# B&R Automation Studio project dbserv_0640 (part 6)

```c
				/* =========================================================== */
				/* DFA-Zustand: Datenobjekt für Datenpunktdefinitionen löschen */
				/* =========================================================== */
				case cCD_PARSER_STATE_DEL_DO_POINT:
					iDatObjDelete.enable = TRUE;
					iDatObjDelete.ident = iDatObjInfo.ident;
					DatObjDelete(&iDatObjDelete);
					if (iDatObjDelete.status == 0) {
						ParserState = cCD_PARSER_STATE_CREATE_DO_POINT;
					}
					else if (iDatObjDelete.status != ERR_FUB_BUSY) {
						ParserState = cCD_PARSER_STATE_ERROR;
					}
					break;

				/* =========================================================== */
				/* DFA-Zustand: Datenobjekt für Datenpunktdefinitionen anlegen */
				/* =========================================================== */
				case cCD_PARSER_STATE_CREATE_DO_POINT:
					iDatObjCreate.enable = TRUE;
					iDatObjCreate.grp = 0;
					iDatObjCreate.pName = (unsigned long)"DpDesc";
					iDatObjCreate.len = countDefinedPoint * sizeof(POINT_DESC);
					iDatObjCreate.MemType = doUSRRAM;
					iDatObjCreate.Option = !doNO_CS;
					iDatObjCreate.pCpyData = (unsigned long)pPointDesc;
					DatObjCreate(&iDatObjCreate);
					if (iDatObjCreate.status == 0) {
						ParserState = cCD_PARSER_STATE_ALLOC_ACCESS_DATA;
					}
					else if (iDatObjCreate.status != ERR_FUB_BUSY) {
						ParserState = cCD_PARSER_STATE_ERROR;
					}
					break;

				/* ======================================= */
				/* DFA-Zustand: Zählen der DBS-Datenpunkte */
				/* ======================================= */
				case cCD_PARSER_STATE_ALLOC_ACCESS_DATA:

					/* --------------------------------------- */
					/* Speicher für Datentypzugriff allokieren */
					/* --------------------------------------- */
					memSize = 0;
					for (i=0; i<=maxDbsUnit; i++) {
						if (pAccessUnit[i].countType > 0) {
							memSize += pAccessUnit[i].countType;
						}
					}
					memSize *= sizeof(ACCESS_TYPE);
					StateTMP_alloc = TMP_alloc(memSize, (void*)&pAccessType);
					if (StateTMP_alloc == 0) {
						SmemSize += 0;
						StmpSize += memSize;
						memset(pAccessType, 0, memSize);

						/* ------------------------------------------ */
						/* Speicher für Anlagenzugriff initialisieren */
						/* ------------------------------------------ */
						pAccessTypeWork = pAccessType;
						for (i=0; i<=maxDbsUnit; i++) {
							if (pAccessUnit[i].countType > 0) {
								pAccessUnit[i].pAccessType = pAccessTypeWork;
								pAccessTypeWork += pAccessUnit[i].countType;
							}
						}

						/* ------------------------------------------- */
						/* Speicher für Datentypzugriff initialisieren */
						/* ------------------------------------------- */
						for (i=0; i<countDefinedPoint; i++) {
							DbsUnit = pPointDesc[i].dbsUnit;
							DbsType = pPointDesc[i].dbsType;
							DbsPoint = pPointDesc[i].dbsPoint;
							pAccessUnit[DbsUnit].pAccessType[DbsType].countPoint = (DbsPoint + 1 > pAccessUnit[DbsUnit].pAccessType[DbsType].countPoint) ? DbsPoint + 1 : pAccessUnit[DbsUnit].pAccessType[DbsType].countPoint;
							pTypeDesc[DbsType].countRelatedPoints++;
						}

						/* ----------------------------------------- */
						/* Speicher für Datenpunktzugriff allokieren */
						/* ----------------------------------------- */
						memSize = 0;
						for (i=0; i<=maxDbsUnit; i++) {
							if (pAccessUnit[i].pAccessType != NULL) {
								for (j=0; j<pAccessUnit[i].countType; j++) {
									memSize += pAccessUnit[i].pAccessType[j].countPoint;
								}
							}
						}
						memSize *= sizeof(ACCESS_POINT);
						StateTMP_alloc = TMP_alloc(memSize, (void*)&pAccessPoint);
						if (StateTMP_alloc == 0) {
							SmemSize += 0;
							StmpSize += memSize;
							memset(pAccessPoint, 0, memSize);

							/* ------------------------------------------- */
							/* Speicher für Datentypzugriff initialisieren */
							/* ------------------------------------------- */
							pAccessPointWork = pAccessPoint;
							for (i=0; i<=maxDbsUnit; i++) {
								for (j=0; j<pAccessUnit[i].countType; j++) {
									if (pAccessUnit[i].pAccessType[j].countPoint > 0) {
										pAccessUnit[i].pAccessType[j].pAccessPoint = pAccessPointWork;
										pAccessPointWork = pAccessPointWork + pAccessUnit[i].pAccessType[j].countPoint;
									}
								}
							}

							/* --------------------------------------------- */
							/* Speicher für Datenpunktzugriff initialisieren */
							/* --------------------------------------------- */
							pAccessDataWork = NULL;
							for (i=0; i<countDefinedPoint; i++) {
								DbsUnit = pPointDesc[i].dbsUnit;
								DbsType = pPointDesc[i].dbsType;
								DbsPoint = pPointDesc[i].dbsPoint;
								countItem = pTypeDesc[DbsType].countItem;
								countTimeItem = pTypeDesc[DbsType].countTimeItem;

								pAccessUnit[DbsUnit].pAccessType[DbsType].pAccessPoint[DbsPoint].pAccessData = pAccessDataWork;
								pAccessTypeWork = &pAccessUnit[DbsUnit].pAccessType[DbsType];
								len = 0;

								pAccessTypeWork->offExtern = len;
								pAccessTypeWork->lenExtern = pTypeDesc[DbsType].sizeType;
								len = pAccessTypeWork->lenExtern;
								if (len % 2 != 0) len++;

								pAccessTypeWork->offIntern = pAccessTypeWork->offExtern + len;
								pAccessTypeWork->lenIntern = pTypeDesc[DbsType].sizeIntType;
								len = pAccessTypeWork->lenIntern;
								if (len % 2 != 0) len++;

								pAccessTypeWork->offiExtern = pAccessTypeWork->offIntern + len;
								pAccessTypeWork->leniExtern = pTypeDesc[DbsType].sizeType;
								pAccessTypeWork->leniExternAlign = (pAccessTypeWork->leniExtern > 1 && pAccessTypeWork->leniExtern % 2 != 0) ? pAccessTypeWork->leniExtern + 1 : pAccessTypeWork->leniExtern;
								pAccessTypeWork->leniExternNext = pAccessTypeWork->leniExternAlign;
								len = countEventInstance * pAccessTypeWork->leniExternAlign;
								if (len % 2 != 0) len++;

								pAccessTypeWork->offValid = pAccessTypeWork->offiExtern + len;
								pAccessTypeWork->lenValid = sizeof(ACCESS_ITEM_VALID);
								pAccessTypeWork->lenValidAlign = (pAccessTypeWork->lenValid > 1 && pAccessTypeWork->lenValid % 2 != 0) ? pAccessTypeWork->lenValid + 1 : pAccessTypeWork->lenValid;
								len = countItem * pAccessTypeWork->lenValidAlign;
								if (len % 2 != 0) len++;

								pAccessTypeWork->offTime = pAccessTypeWork->offValid + len;
								pAccessTypeWork->lenTime = sizeof(RTCtime_typ);
								pAccessTypeWork->lenTimeAlign = (pAccessTypeWork->lenTime > 1 && pAccessTypeWork->lenTime % 2 != 0) ? pAccessTypeWork->lenTime + 1 : pAccessTypeWork->lenTime;
								len = countItem * pAccessTypeWork->lenTimeAlign;
								if (len % 2 != 0) len++;

								pAccessTypeWork->offiTime = pAccessTypeWork->offTime + len;
								pAccessTypeWork->leniTime = sizeof(RTCtime_typ);
								pAccessTypeWork->leniTimeAlign = (pAccessTypeWork->leniTime > 1 && pAccessTypeWork->leniTime % 2 != 0) ? pAccessTypeWork->leniTime + 1 : pAccessTypeWork->leniTime;
								pAccessTypeWork->leniTimeNext = countItem * pAccessTypeWork->leniTimeAlign;
								len = countEventInstance * pAccessTypeWork->leniTimeNext;
								if (len % 2 != 0) len++;

								pAccessTypeWork->offWritelink = pAccessTypeWork->offiTime + len;
								pAccessTypeWork->lenWritelink = sizeof(ACCESS_ITEM_WRITE_LINK);
								pAccessTypeWork->lenWritelinkAlign = (pAccessTypeWork->lenWritelink > 1 && pAccessTypeWork->lenWritelink % 2 != 0) ? pAccessTypeWork->lenWritelink + 1 : pAccessTypeWork->lenWritelink;
								len = countItem * pAccessTypeWork->lenWritelinkAlign;
								if (len % 2 != 0) len++;

								pAccessTypeWork->offWritehandle = pAccessTypeWork->offWritelink + len;
								pAccessTypeWork->lenWritehandle = sizeof(ACCESS_ITEM_WRITE_HANDLE);
								pAccessTypeWork->lenWritehandleAlign = (pAccessTypeWork->lenWritehandle > 1 && pAccessTypeWork->lenWritehandle % 2 != 0) ? pAccessTypeWork->lenWritehandle + 1 : pAccessTypeWork->lenWritehandle;
								len = countItem * pAccessTypeWork->lenWritehandleAlign;
								if (len % 2 != 0) len++;

								pAccessTypeWork->offiEventlink = pAccessTypeWork->offWritehandle + len;
								pAccessTypeWork->leniEventlink = sizeof(ACCESS_ITEM_EVENT_LINK);
								pAccessTypeWork->leniEventlinkAlign = (pAccessTypeWork->leniEventlink > 1 && pAccessTypeWork->leniEventlink % 2 != 0) ? pAccessTypeWork->leniEventlink + 1 : pAccessTypeWork->leniEventlink;
								pAccessTypeWork->leniEventlinkNext = countItem * pAccessTypeWork->leniEventlinkAlign;
								len = countEventInstance * pAccessTypeWork->leniEventlinkNext;
								if (len % 2 != 0) len++;

								pAccessTypeWork->offiReleasestream = pAccessTypeWork->offiEventlink + len;
								pAccessTypeWork->leniReleasestream = sizeof(ACCESS_ITEM_RELEASE);
								pAccessTypeWork->leniReleasestreamAlign = (pAccessTypeWork->leniReleasestream > 1 && pAccessTypeWork->leniReleasestream % 2 != 0) ? pAccessTypeWork->leniReleasestream + 1 : pAccessTypeWork->leniReleasestream;
								pAccessTypeWork->leniReleasestreamNext = countItem * pAccessTypeWork->leniReleasestreamAlign;
								len = countEventInstance * pAccessTypeWork->leniReleasestreamNext;
								if (len % 2 != 0) len++;

								pAccessTypeWork->offiHyst = pAccessTypeWork->offiReleasestream + len;
								pAccessTypeWork->leniHyst = pTypeDesc[DbsType].sizeType;
								pAccessTypeWork->leniHystAlign = (pAccessTypeWork->leniHyst > 1 && pAccessTypeWork->leniHyst % 2 != 0) ? pAccessTypeWork->leniHyst + 1 : pAccessTypeWork->leniHyst;
								pAccessTypeWork->leniHystNext = pAccessTypeWork->leniHystAlign;
								len = countEventInstance * pAccessTypeWork->leniHystNext;
								if (len % 2 != 0) len++;

								pAccessTypeWork->offiEvent = pAccessTypeWork->offiHyst + len;
								pAccessTypeWork->leniEvent = sizeof(ACCESS_ITEM_EVENT_STATE);
								pAccessTypeWork->leniEventAlign = (pAccessTypeWork->leniEvent > 1 && pAccessTypeWork->leniEvent % 2 != 0) ? pAccessTypeWork->leniEvent + 1 : pAccessTypeWork->leniEvent;
								pAccessTypeWork->leniEventNext = countItem * pAccessTypeWork->leniEventAlign;
								len = countEventInstance * pAccessTypeWork->leniEventNext;
								if (len % 2 != 0) len++;

								pAccessTypeWork->offFubInstance = pAccessTypeWork->offiEvent + len;
								pAccessTypeWork->lenFubInstance = sizeof(ACCESS_FUB_INSTANCE);
								pAccessTypeWork->lenFubInstanceAlign = (pAccessTypeWork->lenFubInstance > 1 && pAccessTypeWork->lenFubInstance % 2 != 0) ? pAccessTypeWork->lenFubInstance + 1 : pAccessTypeWork->lenFubInstance;
								len = countItem * pAccessTypeWork->lenFubInstanceAlign;
								if (len % 2 != 0) len++;

								pAccessDataWork = (ACCESS_DATA*)((unsigned char*)pAccessDataWork + pAccessTypeWork->offFubInstance + len);
							} /* (i=0; i<countDefinedPoint; i++) */

							/* ---------------- */
							/* nächster Zustand */
							/* ---------------- */
							ParserState = cCD_PARSER_STATE_COMPARE_DO_DATA;

						} /* (StateTMP_alloc == 0) */
						else {
							/* Fehler bei TMP_alloc */
							ParserState = cCD_PARSER_STATE_ERROR;
						}
					} /* (StateTMP_alloc == 0) */
					else {
						/* Fehler bei TMP_alloc */
						ParserState = cCD_PARSER_STATE_ERROR;
					}
					break;

				/* ==================================== */
				/* DFA-Zustand: Datenobjekt vorhanden ? */
				/* ==================================== */
				case cCD_PARSER_STATE_COMPARE_DO_DATA:
					memSize = (unsigned long)pAccessDataWork;
					if (DbsMemTypeData == 0) {
						StateTMP_alloc = TMP_alloc(memSize, (void*)&pAccessData);
						if (StateTMP_alloc == 0) {
							SmemSize += 0;
							StmpSize += memSize;
							memset(pAccessData, 0, memSize);
							ParserState = cCD_PARSER_STATE_WORK_DATA;
						}
						else {
							ParserState = cCD_PARSER_STATE_ERROR;
						}
					}
					else {
						iDatObjInfo.enable = TRUE;
						iDatObjInfo.pName = (unsigned long)"dbsData";
						DatObjInfo(&iDatObjInfo);
						if (iDatObjInfo.status == 0) {
							/* Datenmodul-Alignment beachten */
							if (iDatObjInfo.len >= memSize &&
								iDatObjInfo.len <  memSize + sizeof(unsigned long) &&
								DbsTypeChanged  == FALSE &&
								DbsPointChanged == FALSE)
							{
								pAccessData = (ACCESS_DATA*)iDatObjInfo.pDatObjMem;
								ParserState = cCD_PARSER_STATE_WORK_DATA;
							}
							else {
								ParserState = cCD_PARSER_STATE_DEL_DO_DATA;
							}
						}
						else if (iDatObjInfo.status == doERR_MODULNOTFOUND) {
							ParserState = cCD_PARSER_STATE_CREATE_DO_DATA;
						}
						else if (iDatObjInfo.status != ERR_FUB_BUSY) {
							ParserState = cCD_PARSER_STATE_ERROR;
						}
					}
					break;

				/* ================================ */
				/* DFA-Zustand: Datenobjekt löschen */
				/* ================================ */
				case cCD_PARSER_STATE_DEL_DO_DATA:
					iDatObjDelete.enable = TRUE;
					iDatObjDelete.ident = iDatObjInfo.ident;
					DatObjDelete(&iDatObjDelete);
					if (iDatObjDelete.status == 0) {
						ParserState = cCD_PARSER_STATE_CREATE_DO_DATA;
					}
					else if (iDatObjDelete.status != ERR_FUB_BUSY) {
						ParserState = cCD_PARSER_STATE_ERROR;
					}
					break;

				/* ==================================== */
				/* DFA-Zustand: Datenobjekt neu anlegen */
				/* ==================================== */
				case cCD_PARSER_STATE_CREATE_DO_DATA:
					iDatObjCreate.enable = TRUE;
					iDatObjCreate.grp = 0;
					iDatObjCreate.pName = (unsigned long)"dbsData";
					iDatObjCreate.len = memSize;
					iDatObjCreate.MemType = doUSRRAM;
					iDatObjCreate.Option = doNO_CS;
					iDatObjCreate.pCpyData = NULL;
					DatObjCreate(&iDatObjCreate);
					if (iDatObjCreate.status == 0) {
						pAccessData = (ACCESS_DATA*)iDatObjCreate.pDatObjMem;
						SmemSize += 0;
						StmpSize += memSize;
						memset(pAccessData, 0, memSize);
						ParserState = cCD_PARSER_STATE_WORK_DATA;
					}
					else if (iDatObjCreate.status != ERR_FUB_BUSY) {
						ParserState = cCD_PARSER_STATE_ERROR;
					}
					break;

				/* ======================================= */
				/* DFA-Zustand: Zählen der DBS-Datenpunkte */
				/* ======================================= */
				case cCD_PARSER_STATE_WORK_DATA:

					/* ------------------------------ */
					/* Pointer auf Datenpunkte setzen */
					/* ------------------------------ */
					for (i=0; i<countDefinedPoint; i++) {
						DbsUnit = pPointDesc[i].dbsUnit;
						DbsType = pPointDesc[i].dbsType;
						DbsPoint = pPointDesc[i].dbsPoint;
						pAccessUnit[DbsUnit].pAccessType[DbsType].pAccessPoint[DbsPoint].pAccessData += (unsigned long)pAccessData;
					}

					/* ---------------------- */
					/* Fubinstanzen eintragen */
					/* ---------------------- */
					for (i=0; i<countFubInstance; i++) {
						DbsUnit = pFubInstanceDesc[i].dbsUnit;
						DbsType = pFubInstanceDesc[i].dbsType;
						DbsPoint = pFubInstanceDesc[i].dbsPoint;
						DbsItem = pFubInstanceDesc[i].dbsItem;
						pAccessTypeWork  = &pAccessUnit[DbsUnit].pAccessType[DbsType];
						pAccessPointWork = &pAccessUnit[DbsUnit].pAccessType[DbsType].pAccessPoint[DbsPoint];
						pAccessFubInstance = (USINT**)(pAccessPointWork->pAccessData + pAccessTypeWork->offFubInstance + DbsItem * pAccessTypeWork->lenFubInstanceAlign);
						*pAccessFubInstance = pFubInstanceDesc[i].pFubInstance;
					}

					/* ---------------- */
					/* nächster Zustand */
					/* ---------------- */
					ParserState = cCD_PARSER_STATE_COMPARE_DO_EVENT;
					break;

				/* ==================================== */
				/* DFA-Zustand: Datenobjekt vorhanden ? */
				/* ==================================== */
				case cCD_PARSER_STATE_COMPARE_DO_EVENT:
					memSize = (maxDbsType + 1) * sizeof(ACCESS_EVENT_PIPE);
					for (i=0; i<=maxDbsType; i++) {
						if (pTypeDesc[i].pItemDesc != NULL && pTypeDesc[i].countRelatedPoints > 0) {
							memSize += countEventInstance * sizeof(EVENT_PIPE_INSTANCE);
							memSize += 	3 * countEventInstance *
										(
											sizeof(EVENT_PIPE_HEADER) +
											(pTypeDesc[i].countRelatedPoints + 1)
											*
											(
												pTypeDesc[i].countItem * sizeof(EVENT_PIPE_DATA) +
												pTypeDesc[i].sizeType +
												pTypeDesc[i].countTimeItem * sizeof(RTCtime_typ)
											)
										);
						}
					}
					if (DbsMemTypeEvent == 0) {
						StateTMP_alloc = TMP_alloc(memSize, (void*)&pEventPipe);
						if (StateTMP_alloc == 0) {
							SmemSize += 0;
							StmpSize += memSize;
							memset(pEventPipe, 0, memSize);
							ParserState = cCD_PARSER_STATE_WORK_EVENT;
						}
						else {
							ParserState = cCD_PARSER_STATE_ERROR;
						}
					}
					else {
						iDatObjInfo.enable = TRUE;
						iDatObjInfo.pName = (unsigned long)"dbsEvent";
						DatObjInfo(&iDatObjInfo);
						if (iDatObjInfo.status == 0) {
							/* Datenmodul-Alignment beachten */
							if (iDatObjInfo.len >= memSize &&
								iDatObjInfo.len <  memSize + sizeof(unsigned long) &&
								DbsTypeChanged  == FALSE &&
								DbsPointChanged == FALSE)
							{
								pEventPipe = (ACCESS_EVENT_PIPE*)iDatObjInfo.pDatObjMem;
								ParserState = cCD_PARSER_STATE_WORK_EVENT;
							}
							else {
								ParserState = cCD_PARSER_STATE_DEL_DO_EVENT;
							}
						}
						else if (iDatObjInfo.status == doERR_MODULNOTFOUND) {
							ParserState = cCD_PARSER_STATE_CREATE_DO_EVENT;
						}
						else if (iDatObjInfo.status != ERR_FUB_BUSY) {
							ParserState = cCD_PARSER_STATE_ERROR;
						}
					}
					break;

				/* ================================ */
				/* DFA-Zustand: Datenobjekt löschen */
				/* ================================ */
				case cCD_PARSER_STATE_DEL_DO_EVENT:
					iDatObjDelete.enable = TRUE;
					iDatObjDelete.ident = iDatObjInfo.ident;
					DatObjDelete(&iDatObjDelete);
					if (iDatObjDelete.status == 0) {
						ParserState = cCD_PARSER_STATE_CREATE_DO_EVENT;
					}
					else if (iDatObjDelete.status != ERR_FUB_BUSY) {
						ParserState = cCD_PARSER_STATE_ERROR;
					}
					break;

				/* ==================================== */
				/* DFA-Zustand: Datenobjekt neu anlegen */
				/* ==================================== */
				case cCD_PARSER_STATE_CREATE_DO_EVENT:
					iDatObjCreate.enable = TRUE;
					iDatObjCreate.grp = 0;
					iDatObjCreate.pName = (unsigned long)"dbsEvent";
					iDatObjCreate.len = memSize;
					iDatObjCreate.MemType = doUSRRAM;
					iDatObjCreate.Option = doNO_CS;
					iDatObjCreate.pCpyData = NULL;
					DatObjCreate(&iDatObjCreate);
					if (iDatObjCreate.status == 0) {
						pEventPipe = (ACCESS_EVENT_PIPE*)iDatObjCreate.pDatObjMem;
						SmemSize += 0;
						StmpSize += memSize;
						memset(pEventPipe, 0, memSize);
						ParserState = cCD_PARSER_STATE_GET_DEVMEMINFO;
					}
					else if (iDatObjCreate.status != ERR_FUB_BUSY) {
						ParserState = cCD_PARSER_STATE_ERROR;
					}
					break;

				/* ==================================== */
				/* DFA-Zustand: Datenobjekt neu anlegen */
				/* ==================================== */
				case cCD_PARSER_STATE_GET_DEVMEMINFO:
					iDevMemInfo.enable = TRUE;
					iDevMemInfo.pDevice = (UDINT)"CompactFlash";
					DevMemInfo(&iDevMemInfo);
					if (iDevMemInfo.status == 0) {
						ParserState = cCD_PARSER_STATE_WORK_EVENT;
					}
					else if (iDevMemInfo.status != ERR_FUB_BUSY) {
						ParserState = cCD_PARSER_STATE_ERROR;
					}
					break;

				/* ==================================== */
				/* DFA-Zustand: Datenobjekt neu anlegen */
				/* ==================================== */
				case cCD_PARSER_STATE_WORK_EVENT:

					/* ---------- */
					/* Event-Pipe */
					/* ---------- */
					memSize = (maxDbsType + 1) * sizeof(ACCESS_EVENT_PIPE);
					for (i=0; i<=maxDbsType; i++) {
						if (pTypeDesc[i].pItemDesc != NULL && pTypeDesc[i].countRelatedPoints > 0) {
							memSize += countEventInstance * sizeof(EVENT_PIPE_INSTANCE);
							memSize += 	3 *	countEventInstance *
										(
											sizeof(EVENT_PIPE_HEADER) +
											(pTypeDesc[i].countRelatedPoints + 1)
											*
											(
												pTypeDesc[i].countItem * sizeof(EVENT_PIPE_DATA) +
												pTypeDesc[i].sizeType +
												pTypeDesc[i].countTimeItem * sizeof(RTCtime_typ)
											)
										);
						}
					} /* (i=0; i<=maxDbsType; i++) */

					StateTMP_alloc = TMP_alloc(memSize, (void*)&pEventPipe);
					if (StateTMP_alloc == 0) {
						SmemSize += 0;
						StmpSize += memSize;
						memset(pEventPipe, 0, memSize);
						pEventPipeInstance = (EVENT_PIPE_INSTANCE*)(pEventPipe + (maxDbsType + 1));

						pEventPipeHeader = (EVENT_PIPE_HEADER*)pEventPipeInstance;
						for (i=0; i<=maxDbsType; i++) {
							if (pTypeDesc[i].pItemDesc != NULL && pTypeDesc[i].countRelatedPoints > 0) {
							//	(USINT*)pEventPipeHeader += countEventInstance * sizeof(EVENT_PIPE_INSTANCE);
/*BIE*/						//	pEventPipeHeader = pEventPipeHeader + countEventInstance * sizeof(EVENT_PIPE_INSTANCE);
								pEventPipeHeader = (EVENT_PIPE_HEADER*)((USINT*)pEventPipeHeader + countEventInstance * sizeof(EVENT_PIPE_INSTANCE));
							}
						}

						for (i=0; i<=maxDbsType; i++) {
							if (pTypeDesc[i].pItemDesc != NULL && pTypeDesc[i].countRelatedPoints > 0) {
								if (pTypeDesc[i].FileBuffer == TRUE) {
									pTypeDesc[i].EventFileBuffer = BufEvents;
									pTypeDesc[i].SizeFileBuffer  = pTypeDesc[i].EventFileBuffer * (sizeof(EVENT_PIPE_DATA) + sizeof(long));
									pTypeDesc[i].ModeFileBuffer  = BufType;
									pEventPipe[i].WriteToFile    = (pTypeDesc[i].SizeFileBuffer > 0) ? TRUE : FALSE;
									pEventPipe[i].SizeFileBuffer = pTypeDesc[i].SizeFileBuffer;
									pEventPipe[i].ModeFileBuffer = pTypeDesc[i].ModeFileBuffer;
								}
								pEventPipe[i].pEventPipeInstance = pEventPipeInstance;

								for (j=0; j<countEventInstance; j++) {
									pEventPipeInstance->pEventPipeHeaderWrite[0] = pEventPipeHeader;
									pEventPipeHeader->pipe_entry = pTypeDesc[i].countRelatedPoints + 1;
									pEventPipeHeader->pipe_size  = pEventPipeHeader->pipe_entry * (	pTypeDesc[i].countItem * sizeof(EVENT_PIPE_DATA) +
																									pTypeDesc[i].sizeType +
																									pTypeDesc[i].countTimeItem * sizeof(RTCtime_typ));
									pEventPipeHeader->pPipeData  = (unsigned char*)&pEventPipeHeader[1];
									pEventPipeHeader->iPipeRead  = 0;
									pEventPipeHeader->iPipeWrite = 0;
									pEventPipeHeader = (EVENT_PIPE_HEADER*)((unsigned char*)pEventPipeHeader->pPipeData + pEventPipeHeader->pipe_size);

									pEventPipeInstance->pEventPipeHeaderWrite[1] = pEventPipeHeader;
									pEventPipeHeader->pipe_entry = pTypeDesc[i].countRelatedPoints + 1;
									pEventPipeHeader->pipe_size  = pEventPipeHeader->pipe_entry * (	pTypeDesc[i].countItem * sizeof(EVENT_PIPE_DATA) +
																									pTypeDesc[i].sizeType +
																									pTypeDesc[i].countTimeItem * sizeof(RTCtime_typ));
									pEventPipeHeader->pPipeData  = (unsigned char*)&pEventPipeHeader[1];
									pEventPipeHeader->iPipeRead  = 0;
									pEventPipeHeader->iPipeWrite = 0;
									pEventPipeHeader = (EVENT_PIPE_HEADER*)((unsigned char*)pEventPipeHeader->pPipeData + pEventPipeHeader->pipe_size);

									pEventPipeInstance->pEventPipeHeaderRead = pEventPipeHeader;
									pEventPipeHeader->pipe_entry = pTypeDesc[i].countRelatedPoints + 1;
									pEventPipeHeader->pipe_size  = pEventPipeHeader->pipe_entry * (	pTypeDesc[i].countItem * sizeof(EVENT_PIPE_DATA) +
																									pTypeDesc[i].sizeType +
																									pTypeDesc[i].countTimeItem * sizeof(RTCtime_typ));
									pEventPipeHeader->pPipeData  = (unsigned char*)&pEventPipeHeader[1];
									pEventPipeHeader->iPipeRead  = 0;
									pEventPipeHeader->iPipeWrite = 0;
									pEventPipeHeader = (EVENT_PIPE_HEADER*)((unsigned char*)pEventPipeHeader->pPipeData + pEventPipeHeader->pipe_size);

									pEventPipeInstance++;
								} /* (j=0; j<countEventInstance; j++) */
							} /* (pTypeDesc[i].pItemDesc != NULL && pTypeDesc[i].countRelatedPoints > 0) */
						} /* (i=0; i<=maxDbsType; i++) */

						/* ---------- */
						/* Write-Pipe */
						/* ---------- */
						memSize = sizeof(ACCESS_WRITE_PIPE) + countWriteInstance * (sizeof(WRITE_PIPE_HEADER) + 64 * (sizeof(WRITE_PIPE_DATA) + sizeof(UDINT)));
						StateTMP_alloc = TMP_alloc(memSize, (void*)&pWritePipe);
						if (StateTMP_alloc == 0) {
							SmemSize += 0;
							StmpSize += memSize;
							memset(pWritePipe, 0, memSize);
							pWritePipeHeader = (WRITE_PIPE_HEADER*)&pWritePipe[1];
							pWritePipe->pWritePipeHeader = pWritePipeHeader;
							for (j=0; j<countWriteInstance; j++) {
								pWritePipeHeader->pipe_entry = 64;
								pWritePipeHeader->pipe_size = pWritePipeHeader->pipe_entry * (sizeof(WRITE_PIPE_DATA) + sizeof(UDINT));
								pWritePipeHeader->pPipeData = (unsigned char*)&pWritePipeHeader[1];
								pWritePipeHeader->iPipeRead = 0;
								pWritePipeHeader->iPipeWrite = 0;
								if (j == 0) {
									pWritePipe->length_pipe_next = sizeof(WRITE_PIPE_HEADER) + pWritePipeHeader->pipe_size;
								}
								pWritePipeHeader = (WRITE_PIPE_HEADER*)((unsigned char*)pWritePipeHeader + pWritePipe->length_pipe_next);
							} /* (j=0; j<countWriteInstance; j++) */

							/* ------------------------------------- */
							/* Speicher für Serverzugriff allokieren */
							/* ------------------------------------- */
							memSize = sizeof(ACCESS_SERVER);
							StateTMP_alloc = TMP_alloc(memSize, (void*)&pAccessServer);
							if (StateTMP_alloc == 0) {
								SmemSize += 0;
								StmpSize += memSize;
								memset(pAccessServer, 0, memSize);

								pAccessServer->countEventInstance = countEventInstance;
								pAccessServer->countWriteInstance = countWriteInstance;
								pAccessServer->countType = maxDbsType + 1;
								pAccessServer->countUnit = maxDbsUnit + 1;
								pAccessServer->pAccessUnit = pAccessUnit;
								pAccessServer->pAccessTypeDesc = pTypeDesc;
								pAccessServer->pAccessPointDesc = pPointDesc;
								pAccessServer->noDevice = cDBS_DEFAULT_DEVICE;
								pAccessServer->pUnitEventState = 0;
								pAccessServer->pAccessEventPipe = pEventPipe;
								pAccessServer->pAccessWritePipe = pWritePipe;
								pAccessServer->PortNumber = PortNumber;
								pAccessServer->TimeoutValue = TimeoutValue;

								idBrServer = pAccessServer;
							}

							/* --------------- */
							/* Logbuch-Ausgabe */
							/* --------------- */
							ultoa((unsigned long) SmemSize / 1024, strcpy(logBuffer, ET_MEM_ALLOC_NEED) + strlen(ET_MEM_ALLOC_NEED));
							ultoa((unsigned long)(SmemSize % 1024 + 50) / 100, strcat(logBuffer,".") + strlen(logBuffer));
							ultoa((unsigned long) StmpSize / 1024, strcat(logBuffer, ET_TMP_ALLOC_NEED) + strlen(logBuffer));
							ultoa((unsigned long)(StmpSize % 1024 + 50) / 100, strcat(logBuffer,".") + strlen(logBuffer));
							strcat(logBuffer, "kB");
							ErrStatistics("dbserv", ERRLOG, 0, 0, ERR_DBS_PRE, logBuffer);

							ultoa((unsigned long)countExistPoints, strcpy(logBuffer, ET_DPS_FOUND) + strlen(ET_DPS_FOUND));
							ultoa((unsigned long)countNotExistPoints, strcat(logBuffer, ET_DPS_NOT_FOUND) + strlen(logBuffer));
							ultoa((unsigned long)countNotExistItems, strcat(logBuffer, ET_ITEM_NOT_FOUND) + strlen(logBuffer));
							if (countInvalidExistItems > 0) {
								strcat(logBuffer, "\n");
								ultoa((unsigned long)countInvalidExistItems, strcat(logBuffer, ET_ITEM_INVALID_FOUND) + strlen(logBuffer));
							}
							ErrStatistics("dbserv", ERRLOG, 0, countNotExistPoints, ERR_DBS_PRE, logBuffer);
							ultoa((unsigned long)BufEvents, strcpy(logBuffer, ET_BUF_EVENTS) + strlen(ET_BUF_EVENTS));
							ErrStatistics("dbserv", ERRLOG, 0, 0, ERR_DBS_PRE, logBuffer);

							/* Berechnung der Speichergrösse für File */
							memSize = (maxDbsType + 1) * sizeof(ACCESS_EVENT_PIPE);
							for (i=0; i<=maxDbsType; i++) {
								if (pTypeDesc[i].pItemDesc != NULL && pTypeDesc[i].countRelatedPoints > 0) {
									memSize += countEventInstance * sizeof(EVENT_PIPE_INSTANCE);
									memSize += countEventInstance *
												(
													sizeof(EVENT_PIPE_HEADER) +
													BufEvents *
													(
														pTypeDesc[i].countItem * sizeof(EVENT_PIPE_DATA) +
														pTypeDesc[i].sizeType +
														pTypeDesc[i].countTimeItem * sizeof(RTCtime_typ)
													)
												);
								}
							}
							ultoa((unsigned long)memSize, strcpy(logBuffer, ET_MEM_EVENTS) + strlen(ET_MEM_EVENTS));
							strcat(logBuffer, "kB");
							ErrStatistics("dbserv", ERRLOG, 0, 0, ERR_DBS_PRE, logBuffer);

							strcat(strcpy(logBuffer, BK_VERSION_TEXT), ET_TCP_READY);
							ErrStatistics("dbserv", ERRLOG, 0, 0, ERR_DBS_PRE, logBuffer);

							/* ---------------- */
							/* nächster Zustand */
							/* ---------------- */
							ParserState = cCD_PARSER_STATE_READY;

						} /* (StateTMP_alloc == 0) */
						else {
							/* Fehler bei TMP_alloc */
							ParserState = cCD_PARSER_STATE_ERROR;
						}
					} /* (StateTMP_alloc == 0) */
					else {
						/* Fehler bei TMP_alloc */
						ParserState = cCD_PARSER_STATE_ERROR;
					}
					break;

			} /* (ParserState) */

			/* ========================================= */
			/* Parser eventuell in Fehlerzustand bringen */
			/* ========================================= */
			/*if (State_find_StationTypPoint < -1 || State_find_Section < -1 || State_find_Data < -1) {*/
			if (State_find_StationTypPoint < -1 || State_find_Section < -1) {
				ParserState = cCD_PARSER_STATE_ERROR;
			}

			/* ======================================== */
			/* Parser in naechsten Zustand schalten ... */
			/* ======================================== */
			switch (ParserState)
			{
/*
				case cCD_PARSER_STATE_DEF_TCP:
					ParserState = cCD_PARSER_STATE_COUNT_TYPE;
					break;

				case cCD_PARSER_STATE_COUNT_TYPE:
					ParserState = cCD_PARSER_STATE_DEF_TYPE;
					break;

				case cCD_PARSER_STATE_DEF_TYPE:
					ParserState = cCD_PARSER_STATE_COMPARE_DO_TYPE;
					break;

				case cCD_PARSER_STATE_COUNT_DP:
					ParserState = cCD_PARSER_STATE_DEF_DP;
					break;

				case cCD_PARSER_STATE_DEF_DP:
					ParserState = cCD_PARSER_STATE_COMPARE_DO_POINT;
					break;

				case cCD_PARSER_STATE_ALLOC_MEM:
					ParserState = cCD_PARSER_STATE_READY;

					ultoa((unsigned long) SmemSize / 1024, strcpy(logBuffer, ET_MEM_ALLOC_NEED) + strlen(ET_MEM_ALLOC_NEED));
					ultoa((unsigned long)(SmemSize % 1024 + 50) / 100, strcat(logBuffer,".") + strlen(logBuffer));
					ultoa((unsigned long) StmpSize / 1024, strcat(logBuffer, ET_TMP_ALLOC_NEED) + strlen(logBuffer));
					ultoa((unsigned long)(StmpSize % 1024 + 50) / 100, strcat(logBuffer,".") + strlen(logBuffer));
					strcat(logBuffer, "kB");
					ErrStatistics(ERRLOG, 0, 0, ERR_DBS_PRE, logBuffer);

					ultoa((unsigned long)countExistPoints, strcpy(logBuffer, ET_DPS_FOUND) + strlen(ET_DPS_FOUND));
					ultoa((unsigned long)countNotExistPoints, strcat(logBuffer, ET_DPS_NOT_FOUND) + strlen(logBuffer));
					ultoa((unsigned long)countNotExistItems, strcat(logBuffer, ET_ITEM_NOT_FOUND) + strlen(logBuffer));
					if (countInvalidExistItems > 0) {
						strcat(logBuffer, "\n");
						ultoa((unsigned long)countInvalidExistItems, strcat(logBuffer, ET_ITEM_INVALID_FOUND) + strlen(logBuffer));
					}
					ErrStatistics(ERRLOG, 0, countNotExistPoints, ERR_DBS_PRE, logBuffer);

					strcat(strcpy(logBuffer, BK_VERSION_TEXT), ET_TCP_READY);
					ErrStatistics(ERRLOG, 0, 0, ERR_DBS_PRE, logBuffer);
					break;
*/
				case cCD_PARSER_STATE_READY:
					CopyPipeToFile(idBrServer);
					break;

				case cCD_PARSER_STATE_ERROR:
					ParserState = cCD_PARSER_STATE_ERROR_READY;
					/* Fehlermeldung */
					if (State_find_StationTypPoint < -1 || State_find_Section < -1 || State_find_Data < -1) {
						strcat(strcpy(logBuffer, (char*)iDatObjInfo.pName), ET_PARSER_STATE);
						if (State_find_StationTypPoint < -1) {
							ultoa(abs(State_find_StationTypPoint), logBuffer + strlen(logBuffer));
						}
						if (State_find_Section < -1) {
							ultoa(abs(State_find_Section), logBuffer + strlen(logBuffer));
						}
						if (State_find_Data < -1) {
							ultoa(abs(State_find_Data), logBuffer + strlen(logBuffer));
						}
						strcat(logBuffer, "\n" );
						sMsgMaxLen = ERRTEXT_MAXLEN - strlen(ERR_DBS_PRE) - 2;
						if (strlen( pParserLine ) > sMsgMaxLen) {
							if (pParserErr - pParserLine > sMsgMaxLen) {
								pParserLine = pParserErr - (sMsgMaxLen * 3) / 4;
							}
						}
						strncat(logBuffer, pParserLine, sMsgMaxLen);
						ErrStatistics("dbserv", ERRLOG, EC_DBS_BASE + EC_PARSER_STATE, CountLines, ERR_DBS_PRE, logBuffer);
					}
					ultoa((unsigned long) SmemSize / 1024, strcpy(logBuffer, ET_MEM_ALLOC_NEED) + strlen(ET_MEM_ALLOC_NEED));
					ultoa((unsigned long)(SmemSize % 1024 + 50) / 100, strcat(logBuffer,".") + strlen(logBuffer));
					ultoa((unsigned long) StmpSize / 1024, strcat(logBuffer, ET_TMP_ALLOC_NEED) + strlen(logBuffer));
					ultoa((unsigned long)(StmpSize % 1024 + 50) / 100, strcat(logBuffer,".") + strlen(logBuffer));
					strcat(logBuffer, "kB");
					ErrStatistics("dbserv", ERRLOG, 0, 0, ERR_DBS_PRE, logBuffer);

					ultoa((unsigned long)countExistPoints, strcpy(logBuffer, ET_DPS_FOUND) + strlen(ET_DPS_FOUND));
					ultoa((unsigned long)countNotExistPoints, strcat(logBuffer, ET_DPS_NOT_FOUND) + strlen(logBuffer));
					ultoa((unsigned long)countNotExistItems, strcat(logBuffer, ET_ITEM_NOT_FOUND) + strlen(logBuffer));
					if (countInvalidExistItems > 0) {
						strcat(logBuffer, "\n");
						ultoa((unsigned long)countInvalidExistItems, strcat(logBuffer, ET_ITEM_INVALID_FOUND) + strlen(logBuffer));
					}
					ErrStatistics("dbserv", ERRLOG, 0, countNotExistPoints, ERR_DBS_PRE, logBuffer);

					strcat(strcpy(logBuffer, BK_VERSION_TEXT), ET_TCP_NOT_READY);
					ErrStatistics("dbserv", ERRLOG, 0, 0, ERR_DBS_PRE, logBuffer);
					break;

				case cCD_PARSER_STATE_ERROR_READY:
					break;

/*
				default:
					ParserState = cCD_PARSER_STATE_ERROR;
					break;
*/

			} /* (ParserState) */
		/*}  (ParserState < cCD_PARSER_STATE_READY) */
	} /* (go == TRUE) */

	/* ------------ */
	/* Testroutinen */
	/* ------------ */
	if (ParserState == cCD_PARSER_STATE_READY) {

		iSysInfo.enable = TRUE;
		SysInfo(&iSysInfo);
		idBrServer->TickCount = iSysInfo.tick_count;

		/* Datentypen */
		pInfoTypeDesc = &pTypeDesc[infoType];
		pInfoItemDesc = pInfoTypeDesc->pItemDesc;
		if (pInfoTypeDesc->pTypeName != NULL) {
			strncpy(InfoTypeName, pInfoTypeDesc->pTypeName, sizeof(InfoTypeName));
		}

		/* Datenpunkte */
		pInfoPointDesc = &pPointDesc[infoPoint];

		SetValueItem (idBrServer,
						1, 1, 33, 0, 0,
						&bValue, sizeof(bValue),
						RTCTime, 0, 1);
	}
} /* _CYCLIC cyclic(void) */

/***********************************************************************/
/* Tcp-Funktionen                                                      */
/***********************************************************************/

unsigned char IsANumber(unsigned char *pData) {

	unsigned char	flag;
	unsigned short	i;

#define	cMAX_CHARACTERS	16

	flag = FALSE;
	if (pData != NULL) {
		for (i=0; i<cMAX_CHARACTERS; i++) {
			if (pData[i] == 0) {
				break;
			}
			else if (pData[i] == ' ' && flag == TRUE) {
				break;
			}
			else if (pData[i]>='0' && pData[i]<='9') {
				flag = TRUE;
			}
			else {
				break;
			}
		}
		if (i == cMAX_CHARACTERS) {
			flag = FALSE;
		}
	}
	return flag;
}

#ifdef x
/*
	ltoa  converts a signed long  value into ASCII Format
	ultoa converts a unsigned long  value into ASCII Format

	both returns the length of the converted string.
*/

int ultoa(unsigned long value, char *buffer) {

	int string_len=0, i, j;
	char swap;

	do {
		buffer[string_len++]=(value % 10) + '0'; /*calculate next digit*/
	} while((value = value/10)); /*while there are more digits*/

	/*swap digits*/
	i=0;
	j=string_len-1;

	while (i<j) {
		swap = buffer[i];
		buffer[i] = buffer[j];
		buffer[j] = swap;
		i++; j--;
	}
	buffer[string_len]=0; /*NULL termination of string*/
	return string_len;    /*Return lenght of string*/
}

int ltoa(long value, char *buffer) {

	int string_len=0, neg=0, i, j;
	char swap;
	unsigned long absval;  /*we have to use unsigned long because, with signed long
	                         0x80000000 would not work.*/

	if (value<0) {
		absval = -value;
		neg=1;
		buffer[0]='-';
		string_len=1;
	}
	else {
		absval = value;
	}
	do {
		buffer[string_len++]=(absval % 10) + '0'; /*calculate next digit*/
	} while((absval = absval/10)); /*while there are more digits*/

	/*swap digits*/
	i=neg;  /*begin at pos 1 if negative*/
	j=string_len-1;

	while (i<j) {
		swap = buffer[i];
		buffer[i] = buffer[j];
		buffer[j] = swap;
		i++; j--;
	}
	buffer[string_len]=0; /*NULL termination of string*/
	return string_len;    /*Return lenght of string*/
}
#endif
/*============================= Ende der Datei ==============================*/
```

### Program Logical/DbServ-Basis/dbsmon (ANSIC, version 6.40.0) - DbServ Monitor

- dbserv.h (reference to Logical/GlobalIncludes/dbserv.h)

#### dbsmon.c
```c
#ifdef _DEFAULT_INCLUDES
	#include <AsDefault.h>
#endif

/******************************************************************************
*    COPYRIGHT    BERNECKER + RAINER Industrie-Elektronik Ges.m.b.H           *
*******************************************************************************
*  Projekt:  DbServ
*  Teil:     Monitor
*  Datei:    bsrun.h
*  Typ:      GNU C (32 Bit)
*------------------------------------------------------------------------------
*  Revision: 01.00
*  Datum:    26-05-2003
*  Autor:    Martin Kurtz / MKrz
*------------------------------------------------------------------------------
*  Funktion: Task-Source-Datei.
*------------------------------------------------------------------------------
*  Rev.  | Datum    | Name | Kommentar
*  ------+----------+------+---------------------------------------------------
*  01.00 | 14-07-03 | MKrz | Modul-Erstellung
*        |          |      |
******************************************************************************/

/***********************************************************************/
/* Headerfiles einbinden                                               */
/***********************************************************************/

#include <bur\plc.h>		/* RPS-spezifische Typendeklarationen */
#include <bur\plctypes.h>	/* RPS-Datentypen */
#include <dataobj.h>		/* SYS_LIB */
#include <sys_lib.h>		/* SYS_LIB */
#include <fileio.h>
#include <string.h>

#include "dbserv.h"

/*************************************************************************************************/
/*	globale Variablen                                                                            */
/*************************************************************************************************/

/*************************************************************************************************/
/*	lokale Variablen                                                                             */
/*************************************************************************************************/
_LOCAL	ACCESS_SERVER	*myidBrServer;
_LOCAL_RETAIN	UINT			statePV_xgetadr	;
static	UDINT			pv_adresse, data_len;

/*
_LOCAL	USINT	*pData_extern, *pData_iextern, *pData_intern, *pData_valid, *pData_time, *pData_itime, *pData_writelink, *pData_ieventlink, *pData_ihyst, *pData_ievent;
_LOCAL	UDINT 	length_extern, length_intern, length_iextern, length_valid, length_time, length_itime, length_writelink, length_ieventlink, length_ihyst, length_ievent;
_LOCAL	UINT	countInstanceAll, countInstanceNoTimestamp, countInstanceTimestamp;
_LOCAL	USINT	tsItem;
_LOCAL	UINT	pipe_entry, pipe_level_abs;
_LOCAL	USINT	pipe_level_rel;
_LOCAL	USINT	bValue;
_LOCAL	UINT	wValue;
_LOCAL	UDINT	lValue;
*/

typedef struct {
	USINT	bValue;
	UINT	wValue;
	UDINT	lValue;
} DATA_VALUE;
/*_LOCAL	DATA_VALUE	DataValue;*/
typedef struct {
	USINT	*pData_extern, *pData_iextern, *pData_intern, *pData_valid, *pData_time, *pData_itime, *pData_writelink, *pData_ieventlink, *pData_ihyst, *pData_ievent;
	UDINT	length_extern, length_intern, length_iextern, length_valid, length_time, length_itime, length_writelink, length_ieventlink, length_ihyst, length_ievent;
} DATA_EXTERN;
/*_LOCAL	DATA_EXTERN	DataExtern;*/
typedef struct {
	UINT	countInstanceAll, countInstanceNoTimestamp, countInstanceTimestamp;
	USINT	tsItem;
} DATA_INSTANCE;
/*_LOCAL	DATA_INSTANCE	DataInstance;*/
typedef struct {
	UINT	pipe_entry, pipe_level_abs;
	USINT	pipe_level_rel;
} DATA_PIPE;
/*_LOCAL	DATA_PIPE	DataPipe;*/
typedef struct {
	UINT			instance;
	UINT			unit;
	UINT			device;
	UINT			type;
	UINT			point;
	UINT			item;
	UINT			infoerror;
	USINT			valid;			/* WAI 18.05.07 */
	DATA_VALUE		DataValue;
	DATA_EXTERN		DataExtern;
	DATA_INSTANCE	DataInstance;
	DATA_PIPE		DataPipe;
} DBS_MONITOR;
_LOCAL_RETAIN	DBS_MONITOR	dbsmon	;

/***********************************************************************************************/
_INIT void init(void)
{
	myidBrServer = NULL;
	statePV_xgetadr = PV_xgetadr("dbserv:idBrServer", &pv_adresse, &data_len);
	if (statePV_xgetadr == 0) {
		myidBrServer = (ACCESS_SERVER*)*(UDINT*)pv_adresse;
	}
} /* _INIT void init(void) */

/***********************************************************************************************/
_CYCLIC	void cyclic(void)
{
	if (myidBrServer == NULL) {

		/* ------------*/
		/* Id-BrServer */
		/* ----------- */
		if (statePV_xgetadr == 0) {
			myidBrServer = (ACCESS_SERVER*)*(UDINT*)pv_adresse;
		}
		else {
			statePV_xgetadr = PV_xgetadr("dbserv:idBrServer", &pv_adresse, &data_len);
		}
	} /* (myidBrServer == NULL) */
	else {

		/* ------------------------ */
		/* Datenpunkt-Informationen */
		/* ------------------------ */
		dbsmon.infoerror = GetItemInfo(myidBrServer, dbsmon.instance,
										dbsmon.unit, dbsmon.device, dbsmon.type, dbsmon.point, dbsmon.item,
										&dbsmon.DataExtern.pData_extern,		&dbsmon.DataExtern.length_extern,
										&dbsmon.DataExtern.pData_intern,		&dbsmon.DataExtern.length_intern,
										&dbsmon.DataExtern.pData_iextern,		&dbsmon.DataExtern.length_iextern,
										&dbsmon.DataExtern.pData_valid,			&dbsmon.DataExtern.length_valid,
										&dbsmon.DataExtern.pData_time,			&dbsmon.DataExtern.length_time,
										&dbsmon.DataExtern.pData_itime,			&dbsmon.DataExtern.length_itime,
										&dbsmon.DataExtern.pData_writelink,		&dbsmon.DataExtern.length_writelink,
										&dbsmon.DataExtern.pData_ieventlink,	&dbsmon.DataExtern.length_ieventlink,
										&dbsmon.DataExtern.pData_ihyst,			&dbsmon.DataExtern.length_ihyst,
										&dbsmon.DataExtern.pData_ievent,		&dbsmon.DataExtern.length_ievent);
		if (dbsmon.infoerror == cEC_OK) {
			switch (dbsmon.DataExtern.length_extern) {
				case 1:
					dbsmon.DataValue.bValue = *(USINT*)dbsmon.DataExtern.pData_extern;
					break;
				case 2:
					dbsmon.DataValue.wValue =  *(UINT*)dbsmon.DataExtern.pData_extern;
					break;
				case 4:
					dbsmon.DataValue.lValue = *(UDINT*)dbsmon.DataExtern.pData_extern;
					break;
			}
			if(dbsmon.DataExtern.pData_valid)	dbsmon.valid = *(dbsmon.DataExtern.pData_valid);
		} /* (infoerror == cEC_OK) */

		/* ------------------ */
		/* Link-Informationen */
		/* ------------------ */
		dbsmon.infoerror = GetEventLinkInfo(myidBrServer,
												dbsmon.unit, dbsmon.device, dbsmon.type, dbsmon.point, dbsmon.item,
												&dbsmon.DataInstance.countInstanceAll,
												&dbsmon.DataInstance.countInstanceNoTimestamp,
												&dbsmon.DataInstance.countInstanceTimestamp,
												&dbsmon.DataInstance.tsItem);

		/* ------------------ */
		/* Pipe-Informationen */
		/* ------------------ */
		GetEventPipeInfo(myidBrServer,
							dbsmon.instance, dbsmon.type,
							&dbsmon.DataPipe.pipe_entry,
							&dbsmon.DataPipe.pipe_level_abs,
							&dbsmon.DataPipe.pipe_level_rel);
	}
} /* _CYCLIC void cyclic(void) */
```

### Program Logical/DbServ-Basis/dbstest (ANSIC, version 6.40.0)

- dbserv.h (reference to Logical/GlobalIncludes/dbserv.h)
